FUNCTION TryConvert_ULINT_TO_DWORD : BOOL
VAR_INPUT
	in : ULINT;
	out : REFERENCE TO DWORD;
END_VAR

IF in > DatatypeLimits.MAX_VALUE_OF_ULINT_WHICH_CAN_BE_HELD_IN_A_DWORD THEN
	RETURN;
END_IF

out := ULINT_TO_DWORD(in);
TryConvert_ULINT_TO_DWORD := TRUE;

END_FUNCTION

(* stored: Version 1.1.0.1, ProductVersion 3.1.4024.12
   POU TryConvert_ULINT_TO_DWORD: Id {34e10ad5-813d-4972-b8ef-a3221a5abb32}, SpecialFunc None *)
